REGION Network 7: Auto run
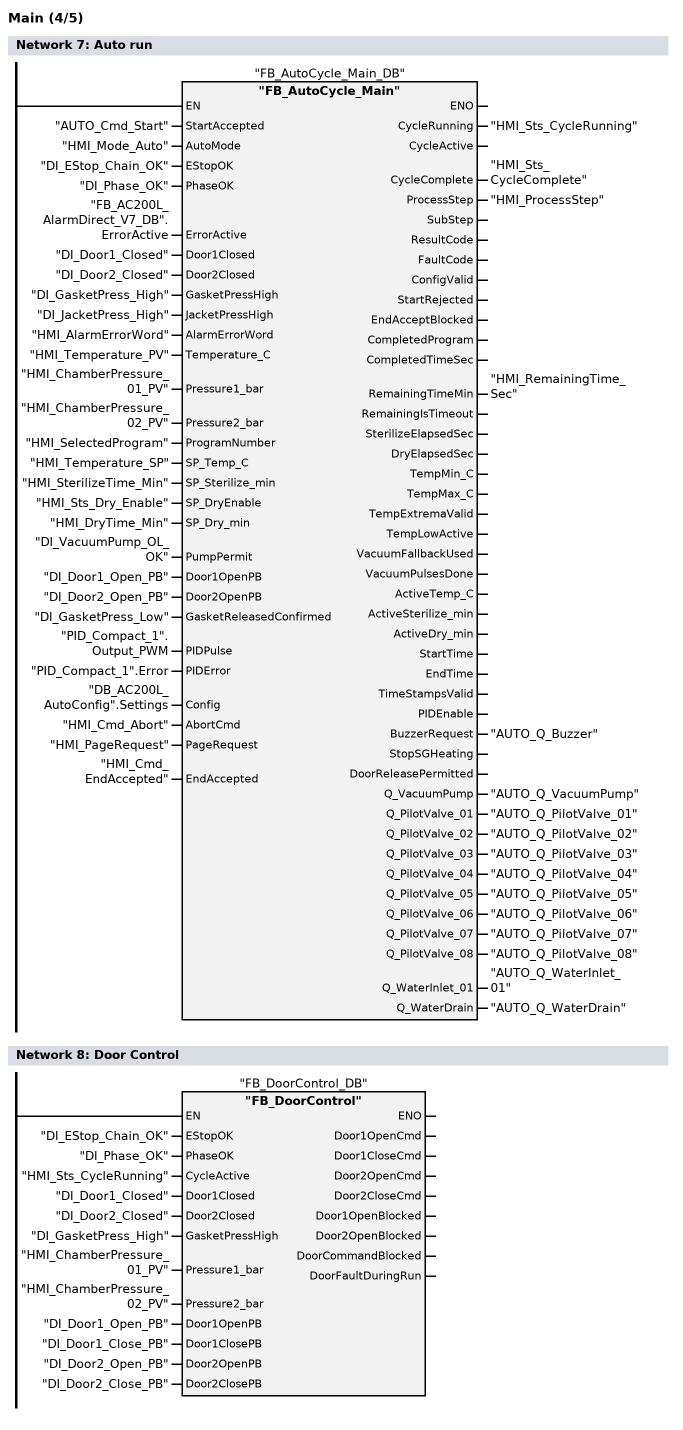
   RUNG wire#powerrail
      "FB_AutoCycle_Main_DB"(StartAccepted := "AUTO_Cmd_Start", AutoMode := "HMI_Mode_Auto", EStopOK := "DI_EStop_Chain_OK", PhaseOK := "DI_Phase_OK", ErrorActive := "FB_AC200L_AlarmDirect_V7_DB".ErrorActive, Door1Closed := "DI_Door1_Closed", Door2Closed := "DI_Door2_Closed", GasketPressHigh := "DI_GasketPress_High", JacketPressHigh := "DI_JacketPress_High", AlarmErrorWord := "HMI_AlarmErrorWord", Temperature_C := "HMI_Temperature_PV", Pressure1_bar := "HMI_ChamberPressure_01_PV", Pressure2_bar := "HMI_ChamberPressure_02_PV", ProgramNumber := "HMI_SelectedProgram", SP_Temp_C := "HMI_Temperature_SP", SP_Sterilize_min := "HMI_SterilizeTime_Min", SP_DryEnable := "HMI_Sts_Dry_Enable", SP_Dry_min := "HMI_DryTime_Min", PumpPermit := "DI_VacuumPump_OL_OK", Door1OpenPB := "DI_Door1_Open_PB", Door2OpenPB := "DI_Door2_Open_PB", GasketReleasedConfirmed := "DI_GasketPress_Low", PIDPulse := "PID_Compact_1".Output_PWM, PIDError := "PID_Compact_1".Error, Config := "DB_AC200L_AutoConfig".Settings, AbortCmd := "HMI_Cmd_Abort", PageRequest := "HMI_PageRequest", EndAccepted := "HMI_Cmd_EndAccepted", CycleRunning => "HMI_Sts_CycleRunning", CycleActive =>, CycleComplete => "HMI_Sts_CycleComplete", ProcessStep => "HMI_ProcessStep", SubStep =>, ResultCode =>, FaultCode =>, ConfigValid =>, StartRejected =>, EndAcceptBlocked =>, CompletedProgram =>, CompletedTimeSec =>, RemainingTimeMin => "HMI_RemainingTime_Sec", RemainingIsTimeout =>, SterilizeElapsedSec =>, DryElapsedSec =>, TempMin_C =>, TempMax_C =>, TempExtremaValid =>, TempLowActive =>, VacuumFallbackUsed =>, VacuumPulsesDone =>, ActiveTemp_C =>, ActiveSterilize_min =>, ActiveDry_min =>, StartTime =>, EndTime =>, TimeStampsValid =>, PIDEnable =>, BuzzerRequest => "AUTO_Q_Buzzer", StopSGHeating =>, DoorReleasePermitted =>, Q_VacuumPump => "AUTO_Q_VacuumPump", Q_PilotValve_01 => "AUTO_Q_PilotValve_01", Q_PilotValve_02 => "AUTO_Q_PilotValve_02", Q_PilotValve_03 => "AUTO_Q_PilotValve_03", Q_PilotValve_04 => "AUTO_Q_PilotValve_04", Q_PilotValve_05 => "AUTO_Q_PilotValve_05", Q_PilotValve_06 => "AUTO_Q_PilotValve_06", Q_PilotValve_07 => "AUTO_Q_PilotValve_07", Q_PilotValve_08 => "AUTO_Q_PilotValve_08", Q_WaterInlet_01 => "AUTO_Q_WaterInlet_01", Q_WaterDrain => "AUTO_Q_WaterDrain")
   END_RUNG
   // the same network as SCL:
   "FB_AutoCycle_Main_DB"(StartAccepted := "AUTO_Cmd_Start",   // "FB_AutoCycle_Main"
                          AutoMode := "HMI_Mode_Auto",
                          EStopOK := "DI_EStop_Chain_OK",
                          PhaseOK := "DI_Phase_OK",
                          ErrorActive := "FB_AC200L_AlarmDirect_V7_DB".ErrorActive,
                          Door1Closed := "DI_Door1_Closed",
                          Door2Closed := "DI_Door2_Closed",
                          GasketPressHigh := "DI_GasketPress_High",
                          JacketPressHigh := "DI_JacketPress_High",
                          AlarmErrorWord := "HMI_AlarmErrorWord",
                          Temperature_C := "HMI_Temperature_PV",
                          Pressure1_bar := "HMI_ChamberPressure_01_PV",
                          Pressure2_bar := "HMI_ChamberPressure_02_PV",
                          ProgramNumber := "HMI_SelectedProgram",
                          SP_Temp_C := "HMI_Temperature_SP",
                          SP_Sterilize_min := "HMI_SterilizeTime_Min",
                          SP_DryEnable := "HMI_Sts_Dry_Enable",
                          SP_Dry_min := "HMI_DryTime_Min",
                          PumpPermit := "DI_VacuumPump_OL_OK",
                          Door1OpenPB := "DI_Door1_Open_PB",
                          Door2OpenPB := "DI_Door2_Open_PB",
                          GasketReleasedConfirmed := "DI_GasketPress_Low",
                          PIDPulse := "PID_Compact_1".Output_PWM,
                          PIDError := "PID_Compact_1".Error,
                          Config := "DB_AC200L_AutoConfig".Settings,
                          AbortCmd := "HMI_Cmd_Abort",
                          PageRequest := "HMI_PageRequest",
                          EndAccepted := "HMI_Cmd_EndAccepted",
                          CycleRunning => "HMI_Sts_CycleRunning",
                          CycleComplete => "HMI_Sts_CycleComplete",
                          ProcessStep => "HMI_ProcessStep",
                          RemainingTimeMin => "HMI_RemainingTime_Sec",
                          BuzzerRequest => "AUTO_Q_Buzzer",
                          Q_VacuumPump => "AUTO_Q_VacuumPump",
                          Q_PilotValve_01 => "AUTO_Q_PilotValve_01",
                          Q_PilotValve_02 => "AUTO_Q_PilotValve_02",
                          Q_PilotValve_03 => "AUTO_Q_PilotValve_03",
                          Q_PilotValve_04 => "AUTO_Q_PilotValve_04",
                          Q_PilotValve_05 => "AUTO_Q_PilotValve_05",
                          Q_PilotValve_06 => "AUTO_Q_PilotValve_06",
                          Q_PilotValve_07 => "AUTO_Q_PilotValve_07",
                          Q_PilotValve_08 => "AUTO_Q_PilotValve_08",
                          Q_WaterInlet_01 => "AUTO_Q_WaterInlet_01",
                          Q_WaterDrain => "AUTO_Q_WaterDrain");
END_REGION

REGION Network 8: Door Control
   RUNG wire#powerrail
      "FB_DoorControl_DB"(EStopOK := "DI_EStop_Chain_OK", PhaseOK := "DI_Phase_OK", CycleActive := "HMI_Sts_CycleRunning", Door1Closed := "DI_Door1_Closed", Door2Closed := "DI_Door2_Closed", GasketPressHigh := "DI_GasketPress_High", Pressure1_bar := "HMI_ChamberPressure_01_PV", Pressure2_bar := "HMI_ChamberPressure_02_PV", Door1OpenPB := "DI_Door1_Open_PB", Door1ClosePB := "DI_Door1_Close_PB", Door2OpenPB := "DI_Door2_Open_PB", Door2ClosePB := "DI_Door2_Close_PB", Door1OpenCmd =>, Door1CloseCmd =>, Door2OpenCmd =>, Door2CloseCmd =>, Door1OpenBlocked =>, Door2OpenBlocked =>, DoorCommandBlocked =>, DoorFaultDuringRun =>)
   END_RUNG
   // the same network as SCL:
   "FB_DoorControl_DB"(EStopOK := "DI_EStop_Chain_OK",   // "FB_DoorControl"
                       PhaseOK := "DI_Phase_OK",
                       CycleActive := "HMI_Sts_CycleRunning",
                       Door1Closed := "DI_Door1_Closed",
                       Door2Closed := "DI_Door2_Closed",
                       GasketPressHigh := "DI_GasketPress_High",
                       Pressure1_bar := "HMI_ChamberPressure_01_PV",
                       Pressure2_bar := "HMI_ChamberPressure_02_PV",
                       Door1OpenPB := "DI_Door1_Open_PB",
                       Door1ClosePB := "DI_Door1_Close_PB",
                       Door2OpenPB := "DI_Door2_Open_PB",
                       Door2ClosePB := "DI_Door2_Close_PB");
END_REGION

REGION Network 9: System Output
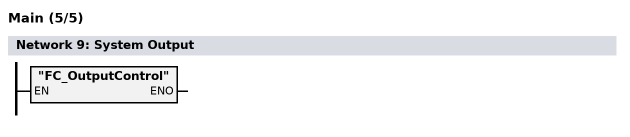
   RUNG wire#powerrail
      "FC_OutputControl"()
   END_RUNG
   // the same network as SCL:
   "FC_OutputControl"();
END_REGION
END_ORGANIZATION_BLOCK

ORGANIZATION_BLOCK "Cyclic interrupt"   // OB30, LAD, CyclicInterrupt
{ S7_Optimized_Access := 'TRUE' }
VERSION : 0.1
   VAR_INPUT
      Initial_Call : Bool;   // Initial call of this OB
      Event_Count : Int;   // Events discarded
   END_VAR
BEGIN

REGION Network 1
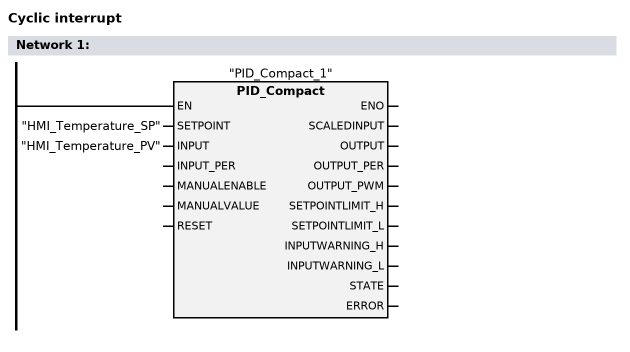
   "PID_Compact_1"(Setpoint := "HMI_Temperature_SP", Input := "HMI_Temperature_PV");   // PID_Compact
END_REGION
END_ORGANIZATION_BLOCK

(* ===== HMI "HMI_RT_1" =====
system functions are stored by id; their names below are inferred from use
connection "HMI_Connection_1": ETHERNET, SMART_S7_1200_OMS

HMI tags "Default tag table"
   "Tag_ScreenNumber" : UInt, internal
   "HMI_AlarmAckWord" : Int = PLC HMI_AlarmAckWord AT %MW172, 1 s

HMI tags "Tag table_manual"
   "HMI_Man_BuzzerTest" : Bool = PLC HMI_Man_BuzzerTest AT %M152.2, 1 s
   "HMI_Man_Heater1" : Bool = PLC HMI_Man_Heater1 AT %M150.2, 1 s
   "HMI_Man_Heater2" : Bool = PLC HMI_Man_Heater2 AT %M150.3, 1 s
   "HMI_Man_Heater3" : Bool = PLC HMI_Man_Heater3 AT %M150.4, 1 s
   "HMI_Man_PilotValve_01" : Bool = PLC HMI_Man_PilotValve_01 AT %M151.0, 1 s
   "HMI_Man_PilotValve_02" : Bool = PLC HMI_Man_PilotValve_02 AT %M151.1, 1 s
   "HMI_Man_PilotValve_03" : Bool = PLC HMI_Man_PilotValve_03 AT %M151.2, 1 s
   "HMI_Man_PilotValve_04" : Bool = PLC HMI_Man_PilotValve_04 AT %M151.3, 1 s
   "HMI_Man_PilotValve_05" : Bool = PLC HMI_Man_PilotValve_05 AT %M151.4, 1 s
   "HMI_Man_PilotValve_06" : Bool = PLC HMI_Man_PilotValve_06 AT %M151.5, 1 s
   "HMI_Man_PilotValve_07" : Bool = PLC HMI_Man_PilotValve_07 AT %M151.6, 1 s
   "HMI_Man_PilotValve_08" : Bool = PLC HMI_Man_PilotValve_08 AT %M151.7, 1 s
   "HMI_Man_VacuumPump" : Bool = PLC HMI_Man_VacuumPump AT %M150.1, 1 s
   "HMI_Man_WaterDrain" : Bool = PLC HMI_Man_WaterDrain AT %M152.1, 1 s
   "HMI_Man_WaterInlet_01" : Bool = PLC HMI_Man_WaterInlet_01 AT %M152.0, 1 s
   "HMI_Man_WaterInlet_02" : Bool = PLC HMI_Man_WaterInlet_02 AT %M152.3, 1 s
   "HMI_Man_WaterPump" : Bool = PLC HMI_Man_WaterPump AT %M150.0, 1 s

HMI tags "Tag table_command"
   "HMI_Cmd_Abort" : Bool = PLC HMI_Cmd_Abort AT %M100.2, 1 s
   "HMI_Cmd_AckAlarm" : Bool = PLC HMI_Cmd_AckAlarm AT %M100.3, 1 s
   "HMI_Cmd_ClearAlarmHistory" : Bool = PLC HMI_Cmd_ClearAlarmHistory AT %M101.5, 1 s
   "HMI_Cmd_Door1Close" : Bool = PLC HMI_Cmd_Door1Close AT %M101.1, 1 s
   "HMI_Cmd_Door1Open" : Bool = PLC HMI_Cmd_Door1Open AT %M101.0, 1 s
   "HMI_Cmd_Door2Close" : Bool = PLC HMI_Cmd_Door2Close AT %M101.3, 1 s
   "HMI_Cmd_Door2Open" : Bool = PLC HMI_Cmd_Door2Open AT %M101.2, 1 s
   "HMI_Cmd_Login" : Bool = PLC HMI_Cmd_Login AT %M101.6, 1 s
   "HMI_Cmd_Logout" : Bool = PLC HMI_Cmd_Logout AT %M101.7, 1 s
   "HMI_Cmd_Print" : Bool = PLC HMI_Cmd_Print AT %M101.4, 1 s
   "HMI_Cmd_Reset" : Bool = PLC HMI_Cmd_Reset AT %M100.4, 1 s
   "HMI_Cmd_Start" : Bool = PLC HMI_Cmd_Start AT %M100.0, 1 s
   "HMI_Cmd_Stop" : Bool = PLC HMI_Cmd_Stop AT %M100.1, 1 s
   "HMI_Mode_Auto" : Bool = PLC HMI_Mode_Auto AT %M100.5, 1 s
   "HMI_Mode_Manual" : Bool = PLC HMI_Mode_Manual AT %M100.6, 1 s
   "HMI_Mode_Service" : Bool = PLC HMI_Mode_Service AT %M100.7, 1 s
   "HMI_Cmd_EndAccepted" : Bool = PLC HMI_Cmd_EndAccepted AT %M121.1, 1 s

HMI tags "Tag table_setpoint"
   "HMI_DryTime_Min" : Int = PLC HMI_DryTime_Min AT %MW108, 1 s
   "HMI_Pressure_SP" : Real = PLC HMI_Pressure_SP AT %MD116, 1 s
   "HMI_PreVacCycles_SP" : Int = PLC HMI_PreVacCycles_SP AT %MW104, 1 s
   "HMI_ProgramNumber" : Int = PLC HMI_ProgramNumber AT %MW102, 1 s
   "HMI_SterilizeTime_Min" : Int = PLC HMI_SterilizeTime_Min AT %MW106, 1 s
   "HMI_Temperature_SP" : Real = PLC HMI_Temperature_SP AT %MD112, 1 s
   "HMI_User_Dry_Min" : Int = PLC HMI_User_Dry_Min AT %MW112, 1 s
   "HMI_User_Temp" : Int = PLC HMI_User_Temp AT %MW114, 1 s
   "HMI_User_Str_Min" : Int = PLC HMI_User_Str_Min AT %MW110, 1 s

HMI tags "Tag table_status"
   "HMI_AlarmErrorWord" : Int = PLC HMI_AlarmErrorWord AT %MW168, 1 s
   "HMI_ChamberPressure_01_PV" : Real = PLC HMI_ChamberPressure_01_PV AT %MD128, 1 s
   "HMI_ChamberPressure_02_PV" : Real = PLC HMI_ChamberPressure_02_PV AT %MD132, 1 s
   "HMI_ProcessStep" : Int = PLC HMI_ProcessStep AT %MW122, 1 s
   "HMI_RemainingTime_Sec" : DInt = PLC HMI_RemainingTime_Sec AT %MD136, 1 s
   "HMI_Sts_AlarmActive" : Bool = PLC HMI_Sts_AlarmActive AT %M120.3, 1 s
   "HMI_Sts_CycleComplete" : Bool = PLC HMI_Sts_CycleComplete AT %M120.2, 1 s
   "HMI_Sts_CycleRunning" : Bool = PLC HMI_Sts_CycleRunning AT %M120.1, 1 s
   "HMI_Sts_Door1Closed" : Bool = PLC HMI_Sts_Door1Closed AT %M120.4, 1 s
   "HMI_Sts_Door2Closed" : Bool = PLC HMI_Sts_Door2Closed AT %M120.5, 1 s
   "HMI_Sts_HeaterRunning" : Bool = PLC HMI_Sts_HeaterRunning AT %M120.6, 1 s
   "HMI_Sts_SystemReady" : Bool = PLC HMI_Sts_SystemReady AT %M120.0, 1 s
   "HMI_Sts_VacuumRunning" : Bool = PLC HMI_Sts_VacuumRunning AT %M120.7, 1 s
   "HMI_Temperature_PV" : Real = PLC HMI_Temperature_PV AT %MD124, 1 s
   "DO_Heater1" : Bool = PLC DO_Heater1 AT %Q0.0, 1 s
   "DO_Heater2" : Bool = PLC DO_Heater2 AT %Q0.1, 1 s
   "DO_Heater3" : Bool = PLC DO_Heater3 AT %Q0.2, 1 s
   "DO_VacuumPump" : Bool = PLC DO_VacuumPump AT %Q0.4, 1 s
   "DO_WaterPump" : Bool = PLC DO_WaterPump AT %Q0.3, 1 s
   "DO_PilotValve_01" : Bool = PLC DO_PilotValve_01 AT %Q8.0, 1 s
   "DO_PilotValve_02" : Bool = PLC DO_PilotValve_02 AT %Q8.1, 1 s
   "DO_PilotValve_03" : Bool = PLC DO_PilotValve_03 AT %Q8.2, 1 s
   "DO_PilotValve_04" : Bool = PLC DO_PilotValve_04 AT %Q8.3, 1 s
   "DO_PilotValve_05" : Bool = PLC DO_PilotValve_05 AT %Q8.4, 1 s
   "DO_PilotValve_06" : Bool = PLC DO_PilotValve_06 AT %Q8.5, 1 s
   "DO_PilotValve_07" : Bool = PLC DO_PilotValve_07 AT %Q8.6, 1 s
   "DO_PilotValve_08" : Bool = PLC DO_PilotValve_08 AT %Q8.7, 1 s
   "DO_WaterInlet_01" : Bool = PLC DO_WaterInlet_01 AT %Q12.0, 1 s
   "DO_WaterInlet_02" : Bool = PLC DO_WaterInlet_02 AT %Q12.6, 1 s
   "DO_WaterDrain" : Bool = PLC DO_WaterDrain AT %Q12.1, 1 s
   "DI_Phase_OK" : Bool = PLC DI_Phase_OK AT %I0.1, 1 s
   "DI_EStop_Chain_OK" : Bool = PLC DI_EStop_Chain_OK AT %I0.0, 1 s
   "DI_Tank_Level_OK" : Bool = PLC DI_Tank_Level_OK AT %I0.4, 1 s
   "DI_SG_Level_High" : Bool = PLC DI_SG_Level_High AT %I0.5, 1 s
   "DI_JacketPress_High" : Bool = PLC DI_JacketPress_High AT %I0.7, 1 s
   "HMI_ChamberPressure_com" : Real = PLC HMI_ChamberPressure_com AT %MD144, 1 s
   "HMI_Sts_Dry_Enable" : Bool = PLC HMI_Sts_Dry_Enable AT %M121.0, 1 s
   "DI_Door1_Closed" : Bool = PLC DI_Door1_Closed AT %I0.2, 1 s
   "DI_Door2_Closed" : Bool = PLC DI_Door2_Closed AT %I0.3, 1 s
   "HMI_AlarmWarningWord" : Int = PLC HMI_AlarmWarningWord AT %MW170, 1 s
   "DI_SGPress_High" : Bool = PLC DI_SGPress_High AT %I1.0, 1 s
   "HMI_StartBlocked" : Bool = PLC HMI_StartBlocked AT %M174.2, 1 s
   "HMI_StartBlockReason" : Int = PLC HMI_StartBlockReason AT %MW174, 1 s
   "AUTO_Cmd_Start" : Bool = PLC AUTO_Cmd_Start AT %M166.1, 1 s
   "HMI_PageRequest" : Int = PLC HMI_PageRequest AT %MW176, 1 s
      on ChangeValue: ActivateScreenByNumber("HMI_PageRequest", 0)
   "HMI_SelectedProgram" : Int = PLC HMI_SelectedProgram AT %MW178, 1 s
   "HMI_ResultCode" : Int = PLC FB_AutoCycle_Demo_DB.ResultCode AT %DB1.DBD0, 1 s

HMI tags "Tag table_time"
   "HMI_Start_Hour" : USInt = PLC FB_AutoCycle_Main_DB.StartTime.HOUR AT %DB1.DBB0, 1 s
   "HMI_Start_Min" : USInt = PLC FB_AutoCycle_Main_DB.StartTime.MINUTE AT %DB1.DBB0, 1 s
   "HMI_Start_Sec" : USInt = PLC FB_AutoCycle_Main_DB.StartTime.SECOND AT %DB1.DBB0, 1 s
   "HMI_End_Hour" : USInt = PLC FB_AutoCycle_Main_DB.EndTime.HOUR AT %DB1.DBB0, 1 s
   "HMI_End_Min" : USInt = PLC FB_AutoCycle_Main_DB.EndTime.MINUTE AT %DB1.DBB0, 1 s
   "HMI_End_Sec" : USInt = PLC FB_AutoCycle_Main_DB.EndTime.SECOND AT %DB1.DBB0, 1 s

discrete alarms
   1: 'Nút dừng khẩn đang tác động', class Errors, trigger "HMI_AlarmErrorWord" bit 0
   2: 'Lỗi nguồn hoặc mất pha', class Errors, trigger "HMI_AlarmErrorWord" bit 1
   3: 'Quá tải bơm nước', class Errors, trigger "HMI_AlarmErrorWord" bit 2
   4: 'Quá tải bơm chân không', class Errors, trigger "HMI_AlarmErrorWord" bit 3
   5: 'Nhiệt độ buồng quá cao', class Errors, trigger "HMI_AlarmErrorWord" bit 4
   6: 'Bồn cấp thiếu nước', class Errors, trigger "HMI_AlarmErrorWord" bit 5
   7: 'Lỗi cảm biến nhiệt độ', class Errors, trigger "HMI_AlarmErrorWord" bit 6
   8: 'Lỗi cảm biến áp suất 1', class Errors, trigger "HMI_AlarmErrorWord" bit 7
   9: 'Lỗi cảm biến áp suất 2', class Errors, trigger "HMI_AlarmErrorWord" bit 8
   10: 'Hai cảm biến áp suất chênh lệch', class Errors, trigger "HMI_AlarmErrorWord" bit 9
   11: 'Quá thời gian ép gioăng', class Errors, trigger "HMI_AlarmErrorWord" bit 10
   12: 'Quá thời gian hút chân không', class Errors, trigger "HMI_AlarmErrorWord" bit 11
   13: 'Quá thời gian gia nhiệt', class Errors, trigger "HMI_AlarmErrorWord" bit 12
   14: 'Nhiệt độ tiệt trùng thấp', class Errors, trigger "HMI_AlarmErrorWord" bit 13
   15: 'Quá thời gian cấp nước bình sinh hơi', class Errors, trigger "HMI_AlarmErrorWord" bit 14
   16: 'Quá thời gian xả áp', class Errors, trigger "HMI_AlarmErrorWord" bit 15
   17: 'Không thể mở cửa khi đang chạy', class Warnings, trigger "HMI_AlarmWarningWord" bit 0
   18: 'Không thể mở cửa khi đang chạy', class Warnings, trigger "HMI_AlarmWarningWord" bit 1
   19: 'Hai cửa chưa đóng an toàn', class Warnings, trigger "HMI_AlarmWarningWord" bit 2
   20: 'Áp suất buồng chưa an toàn để mở cửa (-0.15 < x < 0.15)', class Warnings, trigger "HMI_AlarmWarningWord" bit 3
   21: 'Đến hạn bảo trì', class Warnings, trigger "HMI_AlarmWarningWord" bit 4
   22: 'Mất kết nối HMI', class Warnings, trigger "HMI_AlarmWarningWord" bit 5
   23: 'Máy in có lỗi', class Warnings, trigger "HMI_AlarmWarningWord" bit 6

text list "Text_list_Door": 0 'Open'; 1 'Close'

text list "Text_list_Phase": 0 'Error'; 1 'OK'

text list "Text_list_Water": 0 'Low'; 1 'High'

text list "Text_list_EStop": 1 'Released'; 0 'Pressed'

text list "Text_list_SG": 0 'Not ready'; 1 'Ready'

text list "Text_list_step": 1 'Vacuum'; 2 'Heating'; 3 'Sterilize'; 4 'Exhaust'; 5 'Dry'

text list "Text_list_RUN": 0 'STOPED'; 1 'RUNNING'

text list "Text_list_END Program": 1 'COMPLETED'; 2 'CANCELLED'; 3 'ERROR'

text list "Text_list_programNum": 1 'Unpackaged tools'; 2 'Packaged tools'; 3 'Febric'; 4 'Heavy'; 5 'Light'; 6 'User'; 7 'User'

graphic list "Graphic_list_1": 2 'delete'; 1 'healthy'; 3 'warning'

Template "Template_1" 800x480
   Button "Exit" at 714,429 size 71x50; TextOff 'Exit'; PictureOff "ExitRuntime_KTP700_Basic_PN_TR"; PictureOn "ExitRuntime_KTP700_Basic_PN_TR"
      on Release: StopRuntime(0)
   Button "Log on" at 220,428 size 71x50; TextOff 'Log on'; PictureOff "Login_KTP700_Basic_PN_TR"; PictureOn "Login_KTP700_Basic_PN_TR"
      on Release: function_a2a04561()
   Button "Alarms" at 114,429 size 71x50; TextOff 'Alarms'; PictureOff "AlarmDisplay_KTP700_Basic_PN_TR"; PictureOn "AlarmDisplay_KTP700_Basic_PN_TR"
      on Release: function_ef3f5d25("Alarm window_Pending", -1)
      Appearance <- "HMI_Sts_AlarmActive"
   Button "Start screen" at 14,429 size 71x50; TextOff 'Start screen'; PictureOff "NavigateHome_KTP700_Basic_PN_TR"; PictureOn "NavigateHome_KTP700_Basic_PN_TR"
      on Release: ActivateScreen("Home", 0)

screen "Home" 800x480, template "Template_1"
   on GenerateScreen: SetTag("Tag_ScreenNumber", 1)
   Button "HmiScreenItemData_3" at 320,345 size 160x50; TextOff 'System info'; TextOn 'System'; PictureOff "Navigates to System screens for KTP700 Basic+ PN 15.1.0.0"; PictureOn "Navigates to System screens for KTP700 Basic+ PN 15.1.0.0"; Authorization "Admin_Control"
      on Release: ActivateScreen("System screens", 0)
   Button "HmiScreenItemData_1" at 320,260 size 160x50; TextOn 'Manual test'; TextOff 'Manual test'; PictureOff "hand+interaction+icon-1320165848462055212_32px"; PictureOn "hand+interaction+icon-1320165848462055212_32px"; Authorization "Admin_Control"
      on Release: ActivateScreen("Manual test", 0)
      on Press: SetBit("HMI_Mode_Manual"); ResetBit("HMI_Mode_Auto")
   TextField "HmiScreenItemData_2" at 177,10 size 446x56; Text '200L Central Sterilizer'
   DateTimeField "Date/time field_1" at 684,3 size 110x24
   DateTimeField "Date/time field_2" at 684,30 size 115x29
   Button "HmiScreenItemData_4" at 320,172 size 160x50; TextOn 'Run program'; TextOff 'Run program'; PictureOff "play+player+run+running+start+starting+icon-1320165737084842976_32px"; PictureOn "play+player+run+running+start+starting+icon-1320165737084842976_32px"
      on Release: ActivateScreen("Run program", 0)
      on Press: SetBit("HMI_Mode_Auto"); ResetBit("HMI_Mode_Manual")
   GraphicView "Logo" at 0,3 size 80x77; Picture "logoCIC"
   TextField "Text field_4" at 267,127 size 266x23; Text 'Hello, please select a command.'
   IOField "I/O field_1" at 233,84 size 78x35; FormatPattern 999.99
      ProcessValue <- "HMI_Temperature_PV"
   TextField "Text field_1" at 0,89 size 240x23; Text 'Chamber temperature (°C):'
   TextField "Text field_2" at 329,90 size 163x23; Text 'S.Pressure_1 (bar):'
   IOField "I/O field_2" at 491,84 size 56x35; FormatPattern 99.99
      ProcessValue <- "HMI_ChamberPressure_01_PV"
   IOField "I/O field_3" at 738,84 size 52x35; FormatPattern 99.99
      ProcessValue <- "HMI_ChamberPressure_02_PV"
   TextField "Text field_3" at 576,90 size 163x23; Text 'S.Pressure_2 (bar):'

screen "System screens" 800x480, template "Template_1"
   on GenerateScreen: SetTag("Tag_ScreenNumber", 4)
   Button "Back" at 0,80 size 159x47; TextOff 'Back'
      on Release: ActivateScreen("Home", 0)
   Button "HmiScreenItemData" at 37,164 size 159x47; TextOff 'SIMATIC PLC system diagnos...'; PictureOff "Navigates to SIMATIC PLC system diagnostics for KTP700 Basic+ PN 15.1.0.0"; PictureOn "Navigates to SIMATIC PLC system diagnostics for KTP700 Basic+ PN 15.1.0.0"
      on Release: ActivateScreen("SIMATIC PLC system diagnostics", 0)
   Button "HmiScreenItemData_2" at 37,234 size 159x47; TextOff 'User administration'; PictureOff "Navigates to User administration for KTP700 Basic+ PN 15.1.0.0"; PictureOn "Navigates to User administration for KTP700 Basic+ PN 15.1.0.0"
      on Release: ActivateScreen("User administration", 0)
   Button "HmiScreenItemData_3" at 37,306 size 159x47; TextOff 'System information'; PictureOff "Navigates to System information for KTP700 Basic+ PN 15.1.0.0"; PictureOn "Navigates to System information for KTP700 Basic+ PN 15.1.0.0"
      on Release: ActivateScreen("System information", 0)
   DateTimeField "Date/time field_1" at 685,3 size 103x24
   DateTimeField "Date/time field_2" at 685,30 size 108x24
   GraphicView "Logo" at 0,3 size 80x77; Picture "logoCIC"
   TextField "HmiScreenItemData_1" at 177,10 size 446x56; Text '200L Central Sterilizer'

screen "SIMATIC PLC system diagnostics" 800x480, template "Template_1"
   on GenerateScreen: SetTag("Tag_ScreenNumber", 5)
   SysDiagControl "HmiScreenItemData" at 1,100 size 796x321
   Button "Back" at 1,52 size 159x47; TextOff 'Back'
      on Release: ActivateScreen("System screens", 0)

screen "User administration" 800x480, template "Template_1"
   on GenerateScreen: SetTag("Tag_ScreenNumber", 7)
   UserView "HmiScreenItemData" at 1,100 size 796x321
   Button "Back" at 1,52 size 159x47; TextOff 'Back'
      on Release: ActivateScreen("System screens", 0)

screen "System information" 800x480, template "Template_1"
   on GenerateScreen: SetTag("Tag_ScreenNumber", 8)
   TextField "HmiScreenItemData" at 34,130 size 171x28; Text 'HMI device type:'
   TextField "HmiScreenItemData_1" at 240,130 size 524x28; Text 'KTP700 Basic+ PN 15.1.0.0'
   TextField "HmiScreenItemData_2" at 34,160 size 171x28; Text 'Connection:'
   TextField "HmiScreenItemData_3" at 240,160 size 524x28; Text 'PROFINET (X1)'
   TextField "HmiScreenItemData_4" at 34,190 size 171x28; Text 'PLC:'
   TextField "HmiScreenItemData_5" at 240,190 size 524x28; Text 'SIMATIC S7 1200 CPU 1215 DC/DC/RLY'
   Button "Back" at 0,80 size 159x47; TextOff 'Back'
      on Release: ActivateScreen("System screens", 0)
   TextField "HmiScreenItemData_6" at 177,10 size 446x56; Text '200L Central Sterilizer'
   DateTimeField "Date/time field_1" at 685,3 size 103x24
   DateTimeField "Date/time field_2" at 685,30 size 108x24
   GraphicView "Logo" at 0,3 size 80x77; Picture "logoCIC"

screen "Run program" 800x480
   Button "Start screen" at 14,429 size 71x50; TextOn 'Start screen'; TextOff 'Start screen'; PictureOn "NavigateHome_KTP700_Basic_PN_TR"; PictureOff "NavigateHome_KTP700_Basic_PN_TR"
      on Release: ActivateScreen("Home", 0)
   Button "Exit" at 714,429 size 71x50; TextOn 'Exit'; TextOff 'Exit'; PictureOn "ExitRuntime_KTP700_Basic_PN_TR"; PictureOff "ExitRuntime_KTP700_Basic_PN_TR"
      on Release: StopRuntime(0)
   TextField "Text field_6" at 227,20 size 346x29; Text 'Select the program to operation!'
   Button "Back_1" at 80,100 size 160x120; TextOn 'Unpackaged tools'; TextOff 'Unpackaged tools'; PictureOff "scalpel"; PictureOn "scalpel"
      on Release: SetTag("HMI_ProgramNumber", 1); ActivateScreen("Strating", 0)
   Button "Back_2" at 320,100 size 160x120; TextOn 'Packaged tools'; TextOff 'Packaged tools'; PictureOff "logistics"; PictureOn "logistics"
      on Release: SetTag("HMI_ProgramNumber", 2); ActivateScreen("Strating", 0)
   Button "Back_3" at 80,260 size 160x120; TextOn 'Heavy'; TextOff 'Heavy'; PictureOff "kilogram"; PictureOn "kilogram"
      on Release: SetTag("HMI_ProgramNumber", 4); ActivateScreen("Strating", 0)
   Button "Back_4" at 560,100 size 160x120; TextOn 'Febric'; TextOff 'Febric'; PictureOff "fabric"; PictureOn "fabric"
      on Release: SetTag("HMI_ProgramNumber", 3); ActivateScreen("Strating", 0)
   Button "Back_5" at 320,260 size 160x120; TextOn 'Light'; TextOff 'Light'; PictureOff "lightweight"; PictureOn "lightweight"
      on Release: SetTag("HMI_ProgramNumber", 5); ActivateScreen("Strating", 0)
   Button "Back_6" at 560,260 size 160x120; TextOn 'User'; TextOff 'User'; PictureOff "edit"; PictureOn "edit"
      on Release: SetTag("HMI_ProgramNumber", 6); ActivateScreen("User setting", 0)

screen "Manual test" 800x480
   Button "Start screen" at 14,429 size 71x50; TextOn 'Start screen'; TextOff 'Start screen'; PictureOn "NavigateHome_KTP700_Basic_PN_TR"; PictureOff "NavigateHome_KTP700_Basic_PN_TR"
      on Release: ActivateScreen("Home", 0)
      on Press: ResetBit("HMI_Mode_Manual")
   Button "Exit" at 714,429 size 71x50; TextOn 'Exit'; TextOff 'Exit'; PictureOn "ExitRuntime_KTP700_Basic_PN_TR"; PictureOff "ExitRuntime_KTP700_Basic_PN_TR"
      on Release: StopRuntime(0)
   TextField "Text field_1" at 14,8 size 379x29; Text 'Select the group want to be tested !'
   Button "Back" at 74,90 size 146x68; TextOn 'Back'; TextOff 'Motor'
      on Release: ActivateScreen("Motor", 0)
   Button "Back_1" at 74,195 size 146x68; TextOn 'Back'; TextOff 'Valve'
      on Release: ActivateScreen("Valve", 0)
   Button "Back_2" at 74,300 size 146x68; TextOn 'Back'; TextOff 'Heater'
      on Release: ActivateScreen("Heater", 0)
   Button "Back_3" at 432,355 size 175x38; TextOn 'Back'; TextOff 'BUZZER'
      on Release: InvertBit("HMI_Man_BuzzerTest")
   SymbolicIOField "Symbolic I/O field_1" at 404,116 size 96x32; TextOff '0'; TextOn '1'; TextList "Text_list_Door"
      ProcessValue <- "DI_Door1_Closed"
   TextField "Text field_2" at 340,80 size 170x27; Text 'SYSTEM STATUS'
   TextField "Text field_3" at 340,119 size 64x23; Text 'F.Door:'
   TextField "Text field_4" at 340,172 size 60x23; Text 'Phase:'
   SymbolicIOField "Symbolic I/O field_2" at 404,168 size 96x32; TextOn '1'; TextOff '0'; TextList "Text_list_Phase"
      ProcessValue <- "DI_Phase_OK"
      Appearance <- "DI_Phase_OK"
   TextField "Text field_5" at 527,172 size 65x23; Text 'SGC.W:'
   SymbolicIOField "Symbolic I/O field_3" at 594,168 size 96x32; TextOn '1'; TextOff '0'; TextList "Text_list_Water"
      ProcessValue <- "DI_SG_Level_High"
      Appearance <- "DI_SG_Level_High"
   TextField "Text field_7" at 527,119 size 66x23; Text 'B.Door:'
   SymbolicIOField "Symbolic I/O field_4" at 594,116 size 96x32; TextOn '1'; TextOff '0'; TextList "Text_list_Door"
      ProcessValue <- "DI_Door2_Closed"
   TextField "Text field_8" at 340,225 size 63x23; Text 'E-stop:'
   SymbolicIOField "Symbolic I/O field_5" at 404,220 size 96x32; TextOn '1'; TextOff '0'; TextList "Text_list_EStop"
      ProcessValue <- "DI_EStop_Chain_OK"
      Appearance <- "DI_EStop_Chain_OK"
   TextField "Text field_9" at 340,310 size 310x23; Text 'To try buzzer click the buttom below.'
   TextField "Text field_10" at 527,225 size 49x23; Text 'SG.P:'
   SymbolicIOField "Symbolic I/O field_6" at 594,220 size 96x32; TextOn '1'; TextOff '0'; TextList "Text_list_SG"
      ProcessValue <- "DI_SGPress_High"
      Appearance <- "DI_SGPress_High"
   TextField "Text field_6" at 527,278 size 52x23; Text 'Tank:'
   SymbolicIOField "Symbolic I/O field_7" at 594,272 size 96x32; TextOn '1'; TextOff '0'; TextList "Text_list_Water"
      ProcessValue <- "DI_Tank_Level_OK"
      Appearance <- "DI_Tank_Level_OK"

screen "Motor" 800x480
   Button "Start screen" at 14,429 size 71x50; TextOn 'Start screen'; TextOff 'Start screen'; PictureOn "NavigateHome_KTP700_Basic_PN_TR"; PictureOff "NavigateHome_KTP700_Basic_PN_TR"
      on Release: ActivateScreen("Home", 0)
      on Press: ResetBit("HMI_Mode_Manual")
   Button "Exit" at 714,429 size 71x50; TextOn 'Exit'; TextOff 'Exit'; PictureOn "ExitRuntime_KTP700_Basic_PN_TR"; PictureOff "ExitRuntime_KTP700_Basic_PN_TR"
      on Release: StopRuntime(0)
   Button "Back" at 14,14 size 159x47; TextOn 'Back'; TextOff 'Back'
      on Release: ActivateScreen("Manual test", 0)
   TextField "Text field_1" at 14,77 size 339x23; Text 'Press the button to turn the pump on/off'
   TextField "Text field_2" at 14,107 size 671x23; Text 'Observe the indicator light and sound to check if the device is operating normally.'
   Button "Back_1" at 160,200 size 160x60; TextOn 'Back'; TextOff 'Water pump'
      on Release: InvertBit("HMI_Man_WaterPump")
   Button "Back_2" at 460,200 size 160x60; TextOn 'Back'; TextOff 'Vaccum pump'
      on Release: InvertBit("HMI_Man_VacuumPump")
   Circle "Circle_1" at 216,277 size 48x48
      Appearance <- "DO_WaterPump"
   TextField "Text field_3" at 206,325 size 68x23; Text 'ON/OFF'
   Circle "Circle_2" at 512,277 size 48x48
      Appearance <- "DO_VacuumPump"
   TextField "Text field_4" at 502,325 size 68x23; Text 'ON/OFF'

screen "Valve" 800x480
   Button "Back" at 14,14 size 159x47; TextOn 'Back'; TextOff 'Back'
      on Release: ActivateScreen("Manual test", 0)
   Button "Back_1" at 14,120 size 160x60; TextOn 'Back'; TextOff 'HE Water inlet 1'
      on Release: InvertBit("HMI_Man_WaterInlet_01")
   Circle "Circle_1" at 182,120 size 48x48
      Appearance <- "DO_WaterInlet_01"
   Button "Back_2" at 14,240 size 160x60; TextOn 'Back'; TextOff 'SGC Water inlet 2'
      on Release: InvertBit("HMI_Man_WaterInlet_02")
   Button "Back_3" at 14,360 size 160x60; TextOn 'Back'; TextOff 'Water Drain'
      on Release: InvertBit("HMI_Man_WaterDrain")
   Button "Back_5" at 570,280 size 160x60; TextOn 'Back'; TextOff 'D.valve jacket 7'
      on Release: InvertBit("HMI_Man_PilotValve_07")
   Button "Back_6" at 292,200 size 160x60; TextOn 'Back'; TextOff 'Valve door.S 2'
      on Release: InvertBit("HMI_Man_PilotValve_02")
   Button "Back_7" at 292,280 size 160x60; TextOn 'Back'; TextOff 'Valve chamber 3'
      on Release: InvertBit("HMI_Man_PilotValve_03")
   Button "Back_8" at 292,360 size 160x60; TextOn 'Back'; TextOff 'Valve hepa 4'
      on Release: InvertBit("HMI_Man_PilotValve_04")
   Button "Back_9" at 570,200 size 160x60; TextOn 'Back'; TextOff 'D.valve chamber 6'
      on Release: InvertBit("HMI_Man_PilotValve_06")
   Button "Back_10" at 570,120 size 160x60; TextOn 'Back'; TextOff 'D.valve SGC 5'
      on Release: InvertBit("HMI_Man_PilotValve_05")
   Button "Back_11" at 570,360 size 160x60; TextOn 'Back'; TextOff 'D.valve door.S 8'
      on Release: InvertBit("HMI_Man_PilotValve_08")
   Button "Exit" at 714,429 size 71x50; TextOn 'Exit'; TextOff 'Exit'; PictureOn "ExitRuntime_KTP700_Basic_PN_TR"; PictureOff "ExitRuntime_KTP700_Basic_PN_TR"
      on Release: StopRuntime(0)
   TextField "Text field_1" at 182,12 size 337x23; Text 'Press the button to turn the valve on/off'
   Circle "Circle_2" at 182,240 size 48x48
      Appearance <- "DO_WaterInlet_02"
   Circle "Circle_3" at 182,360 size 48x48
      Appearance <- "DO_WaterDrain"
   Circle "Circle_5" at 738,120 size 48x48
      Appearance <- "DO_PilotValve_05"
   Circle "Circle_6" at 738,200 size 48x48
      Appearance <- "DO_PilotValve_06"
   Circle "Circle_7" at 738,280 size 48x48
      Appearance <- "DO_PilotValve_07"
   Circle "Circle_8" at 738,361 size 48x48
      Appearance <- "DO_PilotValve_08"
   Circle "Circle_4" at 460,120 size 48x48
      Appearance <- "DO_PilotValve_01"
   Button "Back_4" at 292,120 size 160x60; TextOn 'Back'; TextOff 'Valve jacket 1'
      on Release: InvertBit("HMI_Man_PilotValve_01")
   Circle "Circle_9" at 460,200 size 48x48
      Appearance <- "DO_PilotValve_02"
   Circle "Circle_10" at 460,280 size 48x48
      Appearance <- "DO_PilotValve_03"
   Circle "Circle_11" at 460,361 size 48x48
      Appearance <- "DO_PilotValve_04"
   TextField "Text field_2" at 182,38 size 594x23; Text 'Observe the light and sound to check if the device is operating normally.'
   Button "Start screen" at 14,429 size 71x50; TextOn 'Start screen'; TextOff 'Start screen'; PictureOn "NavigateHome_KTP700_Basic_PN_TR"; PictureOff "NavigateHome_KTP700_Basic_PN_TR"
      on Release: ActivateScreen("Home", 0)
      on Press: ResetBit("HMI_Mode_Manual")
   TextField "Text field_3" at 183,64 size 371x23; Text 'Valve 4,5,6,7 and Water Drain are NO valves.'

screen "Heater" 800x480
   Button "Exit" at 714,429 size 71x50; TextOn 'Exit'; TextOff 'Exit'; PictureOn "ExitRuntime_KTP700_Basic_PN_TR"; PictureOff "ExitRuntime_KTP700_Basic_PN_TR"
      on Release: StopRuntime(0)
   Button "Back_1" at 14,14 size 159x47; TextOn 'Back'; TextOff 'Back'
      on Release: ActivateScreen("Manual test", 0)
   TextField "Text field_1" at 14,77 size 428x23; Text 'Press the button to turn the heating element on/off'
   TextField "Text field_2" at 14,107 size 671x23; Text 'Observe the indicator light and sound to check if the device is operating normally.'
   Button "Back_2" at 100,217 size 160x60; TextOn 'Back'; TextOff 'Heater 1'
      on Release: InvertBit("HMI_Man_Heater1")
   Circle "Circle_1" at 156,294 size 48x48
      Appearance <- "DO_Heater1"
   TextField "Text field_3" at 146,342 size 68x23; Text 'ON/OFF'
   TextField "Text field_4" at 14,137 size 551x23; Text 'Caution: The heater ONLY operate when there is water in the SGC.'
   Button "Back_3" at 540,217 size 160x60; TextOn 'Back'; TextOff 'Heater 3'
      on Release: InvertBit("HMI_Man_Heater3")
   Circle "Circle_2" at 596,294 size 48x48
      Appearance <- "DO_Heater3"
   TextField "Text field_5" at 586,342 size 68x23; Text 'ON/OFF'
   Button "Back_4" at 320,217 size 160x60; TextOn 'Back'; TextOff 'Heater 2'
      on Release: InvertBit("HMI_Man_Heater2")
   Circle "Circle_3" at 376,294 size 48x48
      Appearance <- "DO_Heater2"
   TextField "Text field_6" at 366,342 size 68x23; Text 'ON/OFF'
   Button "Start screen" at 14,429 size 71x50; TextOn 'Start screen'; TextOff 'Start screen'; PictureOn "NavigateHome_KTP700_Basic_PN_TR"; PictureOff "NavigateHome_KTP700_Basic_PN_TR"
      on Release: ActivateScreen("Home", 0)
      on Press: ResetBit("HMI_Mode_Manual")

screen "Strating" 800x480, template "Template_2"
   TextField "Text field_1" at 97,16 size 606x29; Text 'Ensure all statuses are displayed in green before starting.'
   Button "Start screen" at 14,429 size 71x50; TextOn 'Start screen'; TextOff 'Start screen'; PictureOn "NavigateHome_KTP700_Basic_PN_TR"; PictureOff "NavigateHome_KTP700_Basic_PN_TR"
      on Release: ActivateScreen("Home", 0)
   Button "Exit" at 714,429 size 71x50; TextOn 'Exit'; TextOff 'Exit'; PictureOn "ExitRuntime_KTP700_Basic_PN_TR"; PictureOff "ExitRuntime_KTP700_Basic_PN_TR"
      on Release: StopRuntime(0)
   Button "Back" at 500,337 size 146x68; TextOn 'Back'; TextOff 'Start'
      on Press: SetBit("HMI_Cmd_Start")
   Button "Back_1" at 154,337 size 146x68; TextOn 'Back'; TextOff 'Cancel'
      on Release: ActivateScreen("Run program", 0)
   SymbolicIOField "Symbolic I/O field_1" at 453,138 size 96x32; TextOn '1'; TextOff '0'; TextList "Text_list_Door"
      ProcessValue <- "DI_Door1_Closed"
      Appearance <- "DI_Door1_Closed"
   TextField "Text field_2" at 389,102 size 170x27; Text 'SYSTEM STATUS'
   TextField "Text field_3" at 389,141 size 64x23; Text 'F.Door:'
   TextField "Text field_4" at 389,194 size 60x23; Text 'Phase:'
   SymbolicIOField "Symbolic I/O field_2" at 453,190 size 96x32; TextOn '1'; TextOff '0'; TextList "Text_list_Phase"
      ProcessValue <- "DI_Phase_OK"
      Appearance <- "DI_Phase_OK"
   TextField "Text field_5" at 576,194 size 65x23; Text 'SGC.W:'
   SymbolicIOField "Symbolic I/O field_3" at 643,190 size 96x32; TextOn '1'; TextOff '0'; TextList "Text_list_Water"
      ProcessValue <- "DI_SG_Level_High"
      Appearance <- "DI_SG_Level_High"
   TextField "Text field_7" at 576,141 size 66x23; Text 'B.Door:'
   SymbolicIOField "Symbolic I/O field_4" at 643,138 size 96x32; TextOn '1'; TextOff '0'; TextList "Text_list_Door"
      ProcessValue <- "DI_Door2_Closed"
      Appearance <- "DI_Door2_Closed"
   TextField "Text field_8" at 389,247 size 63x23; Text 'E-stop:'
   SymbolicIOField "Symbolic I/O field_5" at 453,242 size 96x32; TextOn '1'; TextOff '0'; TextList "Text_list_EStop"
      ProcessValue <- "DI_EStop_Chain_OK"
      Appearance <- "DI_EStop_Chain_OK"
   TextField "Text field_11" at 576,247 size 60x23; Text 'SGC.P:'
   SymbolicIOField "Symbolic I/O field_6" at 642,242 size 96x32; TextOff '0'; TextOn '1'; TextList "Text_list_SG"
      ProcessValue <- "DI_SGPress_High"
      Appearance <- "DI_SGPress_High"
   IOField "I/O field_1" at 210,190 size 96x32; FormatPattern 999
      ProcessValue <- "HMI_DryTime_Min"
   IOField "I/O field_2" at 210,138 size 96x32; FormatPattern 999
      ProcessValue <- "HMI_SterilizeTime_Min"
   IOField "I/O field_3" at 210,242 size 96x32; FormatPattern 999
      ProcessValue <- "HMI_Temperature_SP"
   TextField "Text field_6" at 40,141 size 170x23; Text 'Sterilize time (min):'
   TextField "Text field_9" at 41,194 size 130x23; Text 'Dry time (min):'
   TextField "Text field_10" at 41,247 size 156x23; Text 'Temperature (°C):'
   TextField "Text field_12" at 41,102 size 104x27; Text 'PROGRAM'

screen "Operating" 800x480, template "Template_2"
   Button "Back_1" at 641,429 size 146x50; TextOn 'Back'; TextOff 'Cancel'
      on Release: ActivateScreen("ConfirmAbort", 0)
   TextField "Text field_7" at 24,11 size 141x37; Text 'RUNNING'
      Appearance <- "HMI_Sts_CycleRunning"
   TextField "Text field_2" at 36,71 size 236x29; Text 'Chamber temperature'
   IOField "I/O field_1" at 36,110 size 216x58; FormatPattern 999.99
      ProcessValue <- "HMI_Temperature_PV"
   TextField "Text field_1" at 210,141 size 34x27; Text '°C'
   TextField "Text field_3" at 36,180 size 123x23; Text 'Temp. set point:'
   TextField "Text field_4" at 207,180 size 28x23; Text '°C'
   IOField "I/O field_3" at 155,180 size 56x23; FormatPattern 999.99
      ProcessValue <- "HMI_Temperature_SP"
   TextField "Text field_5" at 36,228 size 134x23; Text 'Chamber pressure'
   IOField "I/O field_2" at 187,246 size 110x33; FormatPattern 99.99
      ProcessValue <- "HMI_ChamberPressure_com"
   TextField "Text field_6" at 292,253 size 42x27; Text 'bar'
   TextField "Text field_8" at 381,65 size 144x29; Text 'Process cycle'
   TextField "Text field_10" at 379,228 size 122x23; Text 'Remaining time:'
   SymbolicIOField "Symbolic I/O field_2" at 459,156 size 222x47; TextOff '0'; TextOn '1'; TextList "Text_list_step"
      ProcessValue <- "HMI_ProcessStep"
   IOField "I/O field_4" at 452,114 size 31x34; FormatPattern 9
      ProcessValue <- "HMI_ProcessStep"
   TextField "Text field_11" at 391,114 size 63x34; Text 'Step:'
   TextField "Text field_12" at 470,114 size 29x34; Text '/5'
   IOField "I/O field_6" at 665,245 size 57x33; FormatPattern 99
      ProcessValue <- "HMI_RemainingTime_Sec"
   TextField "Text field_13" at 36,326 size 96x29; Text 'Program'
   TextField "Text field_20" at 380,325 size 132x27; Text 'System staus'
   TextField "Text field_17" at 381,375 size 73x23; Text 'W.Tank:'
   SymbolicIOField "Symbolic I/O field_1" at 452,373 size 52x29; TextOn '1'; TextOff '0'; TextList "Text_list_Water"
      ProcessValue <- "DI_Tank_Level_OK"
      Appearance <- "DI_Tank_Level_OK"
   TextField "Text field_18" at 519,375 size 60x23; Text 'SGC.P:'
   SymbolicIOField "Symbolic I/O field_4" at 712,373 size 52x29; TextOn '1'; TextOff '0'; TextList "Text_list_Water"
      ProcessValue <- "DI_SGPress_High"
      Appearance <- "DI_SGPress_High"
   TextField "Text field_19" at 648,375 size 65x23; Text 'SGC.W:'
   SymbolicIOField "Symbolic I/O field_3" at 578,373 size 53x29; TextOn '1'; TextOff '0'; TextList "Text_list_Water"
      ProcessValue <- "DI_SG_Level_High"
      Appearance <- "DI_SG_Level_High"
   Group "Group" at 50,375 size 62x23
   Group "Group_1" at 155,375 size 64x23
   Group "Group_2" at 260,375 size 64x23
   TextField "Text field_9" at 713,256 size 47x27; Text 'min'
   TextField "Text field_14" at 83,375 size 29x23; Text '°C'
   IOField "I/O field_5" at 50,375 size 37x23; FormatPattern 999
      ProcessValue <- "HMI_Temperature_SP"
   IOField "I/O field_7" at 155,375 size 30x23; FormatPattern 99
      ProcessValue <- "HMI_SterilizeTime_Min"
   TextField "Text field_15" at 179,375 size 40x23; Text 'min'
   IOField "I/O field_8" at 260,375 size 30x23; FormatPattern 99
      ProcessValue <- "HMI_DryTime_Min"
   TextField "Text field_16" at 284,375 size 40x23; Text 'min'

screen "User setting" 800x480, template "Template_2"
   Button "Start screen" at 14,429 size 71x50; TextOn 'Start screen'; TextOff 'Start screen'; PictureOn "NavigateHome_KTP700_Basic_PN_TR"; PictureOff "NavigateHome_KTP700_Basic_PN_TR"
      on Release: ActivateScreen("Home", 0)
   Button "Exit" at 714,429 size 71x50; TextOn 'Exit'; TextOff 'Exit'; PictureOn "ExitRuntime_KTP700_Basic_PN_TR"; PictureOff "ExitRuntime_KTP700_Basic_PN_TR"
      on Release: StopRuntime(0)
   Button "Back_1" at 145,337 size 146x68; TextOn 'Back'; TextOff 'Cancel'
      on Release: SetTag("HMI_ProgramNumber", 8); ActivateScreen("Run program", 0)
   Button "Back" at 509,337 size 146x68; TextOn 'Back'; TextOff 'Confirm'
      on Release: SetTag("HMI_ProgramNumber", 7); ActivateScreen("Strating", 0)
   TextField "Text field_1" at 223,16 size 334x29; Text 'Selecting operation parameters'
   IOField "I/O field_1" at 420,275 size 96x32; FormatPattern 999
      Appearance <- "HMI_Sts_Dry_Enable"
      ProcessValue <- "HMI_User_Dry_Min"
   IOField "I/O field_2" at 420,175 size 96x32; FormatPattern 999
      ProcessValue <- "HMI_User_Str_Min"
   IOField "I/O field_3" at 420,125 size 96x32; FormatPattern 999
      ProcessValue <- "HMI_User_Temp"
   TextField "Text field_6" at 155,180 size 170x23; Text 'Sterilize time (min):'
   TextField "Text field_9" at 156,280 size 130x23; Text 'Dry time (min):'
   TextField "Text field_10" at 156,130 size 156x23; Text 'Temperature (°C):'
   TextField "Text field_12" at 155,80 size 113x27; Text 'Parameters'
   TextField "Text field_2" at 156,230 size 58x23; Text 'Drying'
   Switch "Switch_1" at 436,225 size 64x32; CaptionText 'Switch'; TextOff 'OFF'; TextOn 'ON'
      on SwitchOn: SetBit("HMI_Sts_Dry_Enable")
      on SwitchOff: ResetBit("HMI_Sts_Dry_Enable")
      Appearance <- "HMI_Sts_Dry_Enable"
      ProcessValue <- "HMI_Sts_Dry_Enable"
   TextField "Text field_3" at 545,130 size 65x23; Text '110-134'
   TextField "Text field_4" at 545,180 size 38x23; Text '1-99'
   TextField "Text field_5" at 545,280 size 38x23; Text '0-99'

screen "ConfirmAbort" 800x480, template "Template_2"
   TextField "Text field_1" at 28,93 size 744x37; Text 'Are you sure you want to cancel the running program?'
   Button "Back" at 500,250 size 146x68; TextOn 'Back'; TextOff 'YES'
      on Release: SetBit("HMI_Cmd_Abort"); ActivateScreen("End screen", 0)
   Button "Back_2" at 154,250 size 146x68; TextOn 'Back'; TextOff 'NO'
      on Release: ActivateScreen("Operating", 0)

screen "End screen" 800x480, template "Template_2"
   SymbolicIOField "Symbolic I/O field_1" at 286,165 size 227x47; TextOff '0'; TextOn '1'; TextList "Text_list_END Program"
      Appearance <- "HMI_Sts_CycleComplete"
      ProcessValue <- "HMI_ResultCode"
   GraphicIOField "Graphic I/O field_1" at 336,20 size 128x128; PictureList "Graphic_list_1"
      ProcessValue <- "HMI_ResultCode"
   Button "Start screen_1" at 290,405 size 220x50; TextOn 'Start screen'; TextOff 'Return home page'; PictureOn "NavigateHome_KTP700_Basic_PN_TR"; PictureOff "NavigateHome_KTP700_Basic_PN_TR"
      on Release: ActivateScreen("Home", 0); SetTag("HMI_PageRequest", 1); SetBit("HMI_Cmd_EndAccepted")
   TextField "Text field_2" at 176,245 size 104x32; Text 'Program'
   SymbolicIOField "Symbolic I/O field_2" at 112,310 size 232x32; TextOff '0'; TextOn '1'; TextList "Text_list_programNum"
      ProcessValue <- "HMI_SelectedProgram"
   TextField "Text field_3" at 540,245 size 62x32; Text 'Time'
   Group "Group" at 460,285 size 223x32
   Group "Group_1" at 460,335 size 223x32
   TextField "Text field_5" at 460,335 size 56x32; Text 'End:'
   IOField "I/O field_4" at 541,335 size 32x32; FormatPattern 99
      ProcessValue <- "HMI_End_Hour"
   TextField "Text field_7" at 577,335 size 13x29; Text ':'
   IOField "I/O field_5" at 596,335 size 32x32; FormatPattern 99
      ProcessValue <- "HMI_End_Min"
   TextField "Text field_9" at 633,335 size 13x29; Text ':'
   IOField "I/O field_6" at 651,335 size 32x32; FormatPattern 99
      ProcessValue <- "HMI_End_Sec"
   IOField "I/O field_3" at 540,285 size 33x32; FormatPattern 99
      ProcessValue <- "HMI_Start_Hour"
   TextField "Text field_6" at 577,285 size 13x29; Text ':'
   TextField "Text field_4" at 460,285 size 72x32; Text 'Start:'
   IOField "I/O field_1" at 595,285 size 33x32; FormatPattern 99
      ProcessValue <- "HMI_Start_Min"
   IOField "I/O field_2" at 650,285 size 33x32; FormatPattern 99
      ProcessValue <- "HMI_Start_Sec"
   TextField "Text field_8" at 633,285 size 13x29; Text ':'
*)